FUNCTION_BLOCK FB_SEL_INT (* INT Selection *)
  (* Standard: 61499-1 *)
  (* Version 0.0, 2001-04-04, JHC, Rockwell Automation, Algorithm in ST *)
  (* Compiler header: package fb.rt.omac; *)
  (* Compiler Java IBM Jikes 1.06 *)
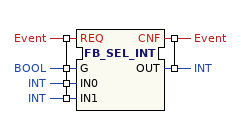
  EVENT_INPUT
    REQ WITH G, IN0, IN1;
  END_EVENT
  EVENT_OUTPUT
    CNF WITH OUT;
  END_EVENT
  VAR_INPUT
    G : BOOL; (* Selector *)
    IN0 : INT; (* Selected when G=0 *)
    IN1 : INT; (* Selected when G=1 *)
  END_VAR
  VAR_OUTPUT
    OUT : INT; (* Selected value *)
  END_VAR
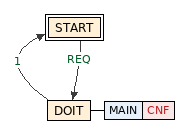
  EC_STATES
    START;
    DOIT : MAIN -> CNF;
  END_STATES
  EC_TRANSITIONS
    START TO DOIT := REQ;
    DOIT TO START := 1;
  END_TRANSITIONS
  ALGORITHM MAIN IN ST:
IF G THEN OUT:=IN1;
ELSE OUT:=IN0;
END_IF
  END_ALGORITHM
END_FUNCTION_BLOCK
